FUNCTION_BLOCK CM_DoorLock EXTENDS CM_Base //--IMPLEMENTS I_Door
VAR
	// Inputs
	I_bStaDoorIsClosed AT %I* : BOOL; // Door is closed
	I_bStaDoorIsReleased AT %I* : BOOL; // Door is released
	I_bPbUnlockDoor AT %I* : BOOL; // Request to unlock door
	
	// Outputs
	Q_bCmdRelease AT %Q* : BOOL; // FALSE = Apply, TRUE = Release
	Q_bStaLamp AT %Q* : BOOL; //Status: OFF = Applied (Locked), ON = Released, FLASHING = Request pending
			
	// Requests
	s_bReqReleaseLock : BOOL;
	s_bReqApplyLock : BOOL;
	
	// States
	s_bStaReqReleaseLock : BOOL;
	s_bStaDoorIsClosed : BOOL;
	s_bStaLockIsApplied : BOOL;
	s_bStaLockIsReleased : BOOL;
	
	// Timers
	fbFlash : FB_Flash;
	
	// Alarms
	s_fbAlarmHandlerDoorNotClosed : FB_AlarmHandler;
	s_fbAlarmHandlerRequestPending : FB_AlarmHandler;
	
	s_wrnDoorNotClosed : BOOL;
	s_infRequestPending : BOOL;
	
	// Toggele request to release door lock
	fbToggleReleaseRequest : FB_Toggle;
	
END_VAR


SUPER^();

METHOD PROTECTED _m_Alarms : BOOL

IF NOT SUPER^._m_Alarms() THEN
	RETURN;
END_IF

// Set error bits
//..

// Alarm Handlers
s_fbAlarmHandlerDoorNotClosed(
	i_bStaActive := s_wrnDoorNotClosed, 
	i_eAlarmLevel := E_AlarmLevel.Warning,
	i_sAlarmText := CONCAT(i_sCmName , CONCAT(': Door - ', 'Apply lock not allowed (close door first).')) );
	
s_fbAlarmHandlerRequestPending(
	i_bStaActive := s_infRequestPending, 
	i_eAlarmLevel := E_AlarmLevel.Info,
	i_sAlarmText := CONCAT(i_sCmName , CONCAT(': Door - ', 'Request to unlock door pending (please wait...).')) );
	
// Alarm collector	
s_bStaError := FALSE;

_m_Alarms := TRUE;
END_METHOD

METHOD PROTECTED _m_Devices : BOOL

IF NOT SUPER^._m_Devices() THEN
	RETURN;
END_IF

IF s_bStaDoorIsClosed THEN
	s_wrnDoorNotClosed := FALSE;
END_IF

IF s_bStaLockIsReleased THEN
	s_infRequestPending := FALSE;
END_IF

//--// Reset request
//--IF s_bStaLockIsReleased THEN
//--	s_bReqReleaseLock := FALSE;
//--ELSIF s_bStaLockIsApplied THEN
//--	s_bReqApplyLock := FALSE;	
//--ELSIF s_bStaError THEN
//--	s_bReqReleaseLock := FALSE;
//--	s_bReqApplyLock := FALSE;
//--END_IF

_m_Devices := TRUE;
END_METHOD

METHOD PROTECTED _m_Hmi : BOOL

IF NOT SUPER^._m_Hmi() THEN
	RETURN;
END_IF

_m_Hmi := TRUE;
END_METHOD

METHOD PROTECTED _m_Init : BOOL

IF NOT SUPER^._m_Init() THEN
	RETURN;
END_IF

{warning '#TODO: Not sure if this control module needs initialzation'}
//--s_DOValve.i_stSettings.bCfgDelay 		:= FALSE;
//--s_DOValve.i_stSettings.tmOutputDelay 	:= T#0S;

_m_Init := TRUE;
END_METHOD

METHOD PROTECTED _m_Inputs : BOOL

IF NOT SUPER^._m_Inputs() THEN
	RETURN;
END_IF

fbToggleReleaseRequest(CLK := I_bPbUnlockDoor);
s_bStaReqReleaseLock := fbToggleReleaseRequest.Q;

s_bStaLockIsReleased := I_bStaDoorIsReleased;
s_bStaLockIsApplied := NOT(I_bStaDoorIsReleased);
s_bStaDoorIsClosed := I_bStaDoorIsClosed;

_m_Inputs := TRUE;
END_METHOD

METHOD PROTECTED _m_Outputs : BOOL

IF NOT SUPER^._m_Outputs() THEN
	RETURN;
END_IF

// Generate flashing pulse for blinking request pending lamp
fbFlash(
	i_bExcecute := s_bStaReqReleaseLock,
	t_tOnTime := T#500MS,
	t_tOffTime := T#1000MS);

Q_bCmdRelease := s_bReqReleaseLock;
Q_bStaLamp := fbFlash.o_bQ; 
	
_m_Outputs := TRUE;
END_METHOD

/// Request to apply door-lock (only if door is closed)
METHOD PUBLIC m_Apply : BOOL

IF NOT i_bReqEnable THEN 
	RETURN;
END_IF

IF s_bStaDoorIsClosed THEN
	s_bReqReleaseLock := FALSE;
	s_bReqApplyLock := TRUE;
ELSE
	s_wrnDoorNotClosed := TRUE;
END_IF
	
m_Apply := TRUE;
END_METHOD

/// Request to release door-lock
METHOD PUBLIC m_Release : BOOL

IF NOT i_bReqEnable THEN 
	RETURN;
END_IF

s_bReqReleaseLock := TRUE;
s_bReqApplyLock := FALSE;

s_infRequestPending := TRUE;

m_Release := TRUE;
END_METHOD

{attribute 'monitoring':='call'}
PROPERTY PUBLIC p_bReqReleaseLock : BOOL
GET

p_bReqReleaseLock := s_bStaReqReleaseLock;
END_GET
END_PROPERTY

{attribute 'monitoring':='call'}
PROPERTY PUBLIC p_bStaDoorIsClosed : BOOL
GET

p_bStaDoorIsClosed := s_bStaDoorIsClosed;
END_GET
END_PROPERTY

{attribute 'monitoring':='call'}
PROPERTY PUBLIC p_bStaLockIsApplied : BOOL
GET

p_bStaLockIsApplied := s_bStaLockIsApplied;
END_GET
END_PROPERTY

{attribute 'monitoring':='call'}
PROPERTY PUBLIC p_bStaLockIsReleased : BOOL
GET

p_bStaLockIsReleased := s_bStaLockIsReleased;
END_GET
END_PROPERTY

END_FUNCTION_BLOCK

(* stored: Version 1.1.0.1, ProductVersion 3.1.4024.12
   POU CM_DoorLock: Id {ea68c333-cb10-44e9-998f-ee97a6acb23c}, SpecialFunc None
   Folder Methods: Id {f1e13262-5093-4e19-b253-1c3417c042de}
   Folder Properties: Id {1cd224f2-8e0f-4515-bca2-e2383476522d}
   Method _m_Alarms: Id {9c548875-33a6-42e4-a316-602892fa3d9c}
   Method _m_Devices: Id {610e92a2-55de-4c20-9dc9-5d6693ddaa6b}
   Method _m_Hmi: Id {099a1203-e422-4fa7-896f-2cb9acc72e21}
   Method _m_Init: Id {7e974ef6-a453-4752-8fef-bd0c78d3fc41}
   Method _m_Inputs: Id {0f80ea41-d213-4e61-bf55-0e2eaf7e039c}
   Method _m_Outputs: Id {505e11af-7bdd-44b3-8506-0a1a26a8e0b6}
   Method m_Apply: Id {1802c1c5-3d52-4491-b19a-2db94b292512}
   Method m_Release: Id {4b2987be-5b37-448a-ae60-0d85428f41cd}
   Property p_bReqReleaseLock: Id {085fa38b-af4e-4f0c-a85b-311bf38ba91d}
   Get Get: Id {c892ec1b-d93f-48c3-bfe3-815a2bf64387}
   Property p_bStaDoorIsClosed: Id {6fc03739-dce9-4ee2-80bf-9e9172243c54}
   Get Get: Id {0a1b8b1e-e1eb-426d-a4e4-2cee32698ff0}
   Property p_bStaLockIsApplied: Id {30b69388-1c5c-4cc9-9c25-d58f841ab12c}
   Get Get: Id {2cd3b54e-5a1b-4a83-a32c-e86b48816fb2}
   Property p_bStaLockIsReleased: Id {ace57d84-4ff8-4d03-a4df-c730a29a90b7}
   Get Get: Id {25e3e480-7e08-4443-a7b7-3684820a84de} *)
